(* Logix 5000 project; controller cal1632 1756-L62 rev 16.20; software revision 16.05; part 17 of 61 *)
(* tags used below, declared in another part *)
   FAULT : BOOL;
   p01_param_oven_timer_presets : DINT[32];
   p01_param_process_air_hl : REAL;
   p01_sys_enc : SYS_ENC;
   p01_sys_lc : Limit_Clamp;
   p01r09_pb_global_reset : BOOL;
   p02_real_from_hmi : hmi_real;
   p12_di_burner_auto : BOOL;
   p12_di_burner_safeties_ok : BOOL;
   p12_di_exh_flow_ok : BOOL;
   p12_di_flame_on : BOOL;
   p12_di_recirc_flow_ok : BOOL;
   p12_dint_to_hmi : DINT[16];
   p12_param_fast_to_soak : REAL;
   p12_param_lfl_hhl : REAL;
   p12_param_lfl_hl : REAL;
   p12_param_pid1_ff : REAL;
   p12_param_pid1_kd : REAL;
   p12_param_pid1_ki : REAL;
   p12_param_pid1_kp : REAL;
   p12_param_pid2_ff : REAL;
   p12_param_pid2_kd : REAL;
   p12_param_pid2_ki : REAL;
   p12_param_pid2_kp : REAL;
   p12_param_shutdown_temp : REAL;
   p12_param_soak_to_fast : REAL;
   p12_param_tc01_dev : REAL;
   p12_param_tc01_hl : REAL;
   p12_param_tc01z : REAL;
   p12_param_tc02z : REAL;
   p12_param_zone_pressure : REAL;
   p12r02 : routine;
   p12r02_shutdown_temp : BOOL;
   p12r02_timer_safe_temp : TIMER[2];
   p12r02_timer_warning : TIMER[4];
   p12r08 : routine;
   p12r08_timer_fault : TIMER[4];
   p12r08_timer_warning : TIMER[4];
   p12r09 : routine;
   p12r09_timer_fault : TIMER[4];
   p12r09_timer_warning : TIMER[8];
   p12r10 : routine;
   p12r10_timer_fault : TIMER[4];
   p12r10_timer_warning : TIMER[4];
   p12r20 : routine;
   p12r20_safeties_ok : BOOL;
   p12r20_state : DINT;
   p12r20_status : DINT;
   p12r20_timer_fault : TIMER[4];
   p12r20_timer_state_11 : TIMER;
   p12r20_timer_state_3 : TIMER;
   p12r20_timer_state_4 : TIMER;
   p12r20_timer_state_7 : TIMER;
   p12r20_timer_warning : TIMER[4];
   p12r30 : routine;
   p12r30_cv_man_sp : REAL;
   p12r30_request_heat : BOOL;
   p12r30_request_manual : BOOL;
   p12r30_request_soak_control : BOOL;
   p12r30_temp_deviation_setpoint : DINT;
   p12r30_timer_fault : TIMER[16];
   p12r30_timer_warning : TIMER[12];
   p12r31 : routine;
   p12r31_timer_fault : TIMER[5];
   p12r31_timer_warning : TIMER[5];
   p12r32 : routine;
   p12r32_timer_fault : TIMER[5];
   p12r32_timer_warning : TIMER[5];
(* P12_Zone_2, continued *)

ROUTINE R08_Warnings   (* ladder *)
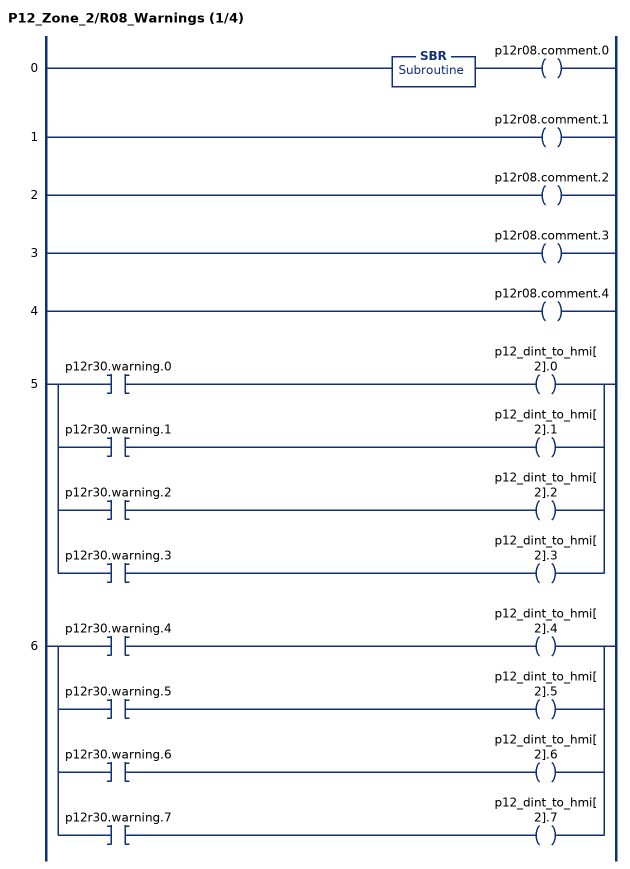
   0: SBR()OTE(p12r08.comment.0);
   1: OTE(p12r08.comment.1);
   2: OTE(p12r08.comment.2);
   3: OTE(p12r08.comment.3);
   4: OTE(p12r08.comment.4);
   5: [XIC(p12r30.warning.0) OTE(p12_dint_to_hmi[2].0) ,XIC(p12r30.warning.1) OTE(p12_dint_to_hmi[2].1) ,XIC(p12r30.warning.2) OTE(p12_dint_to_hmi[2].2) ,XIC(p12r30.warning.3) OTE(p12_dint_to_hmi[2].3) ];
   6: [XIC(p12r30.warning.4) OTE(p12_dint_to_hmi[2].4) ,XIC(p12r30.warning.5) OTE(p12_dint_to_hmi[2].5) ,XIC(p12r30.warning.6) OTE(p12_dint_to_hmi[2].6) ,XIC(p12r30.warning.7) OTE(p12_dint_to_hmi[2].7) ];
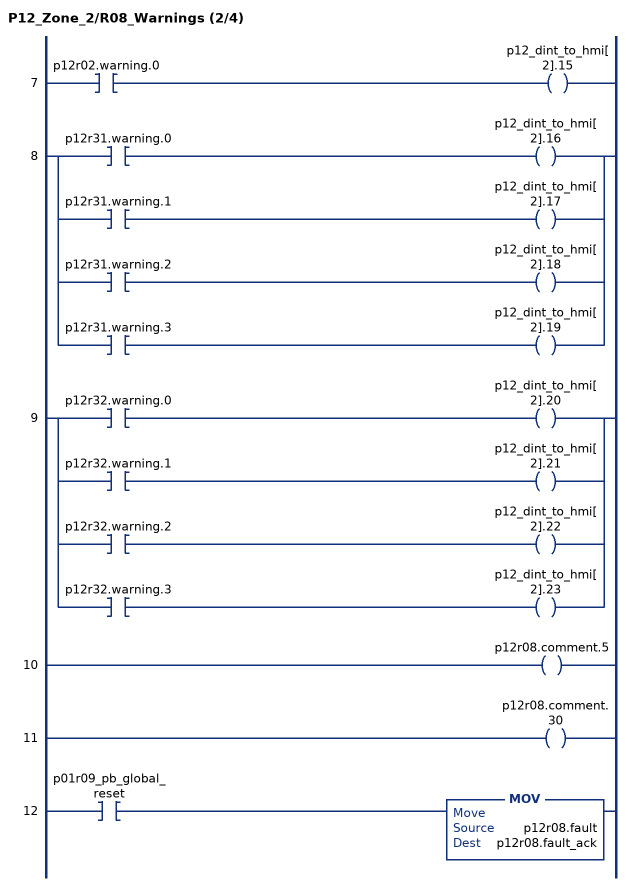
   7: XIC(p12r02.warning.0)OTE(p12_dint_to_hmi[2].15);
   8: [XIC(p12r31.warning.0) OTE(p12_dint_to_hmi[2].16) ,XIC(p12r31.warning.1) OTE(p12_dint_to_hmi[2].17) ,XIC(p12r31.warning.2) OTE(p12_dint_to_hmi[2].18) ,XIC(p12r31.warning.3) OTE(p12_dint_to_hmi[2].19) ];
   9: [XIC(p12r32.warning.0) OTE(p12_dint_to_hmi[2].20) ,XIC(p12r32.warning.1) OTE(p12_dint_to_hmi[2].21) ,XIC(p12r32.warning.2) OTE(p12_dint_to_hmi[2].22) ,XIC(p12r32.warning.3) OTE(p12_dint_to_hmi[2].23) ];
   10: OTE(p12r08.comment.5);
   11: OTE(p12r08.comment.30);
   12: XIC(p01r09_pb_global_reset)MOV(p12r08.fault,p12r08.fault_ack);
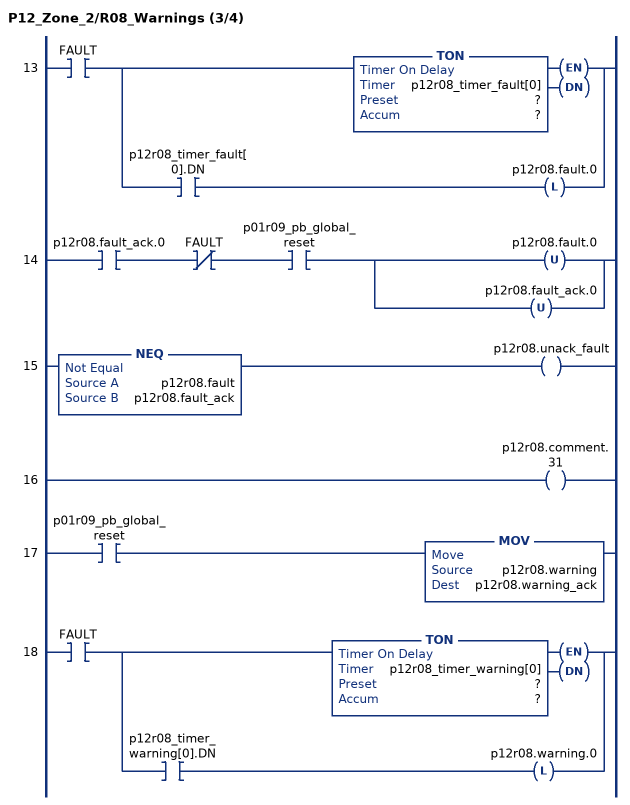
   13: XIC(FAULT)[TON(p12r08_timer_fault[0],?,?) ,XIC(p12r08_timer_fault[0].DN) OTL(p12r08.fault.0) ];
   14: XIC(p12r08.fault_ack.0)XIO(FAULT)XIC(p01r09_pb_global_reset)[OTU(p12r08.fault.0) ,OTU(p12r08.fault_ack.0) ];
   15: NEQ(p12r08.fault,p12r08.fault_ack)OTE(p12r08.unack_fault);
   16: OTE(p12r08.comment.31);
   17: XIC(p01r09_pb_global_reset)MOV(p12r08.warning,p12r08.warning_ack);
   18: XIC(FAULT)[TON(p12r08_timer_warning[0],?,?) ,XIC(p12r08_timer_warning[0].DN) OTL(p12r08.warning.0) ];
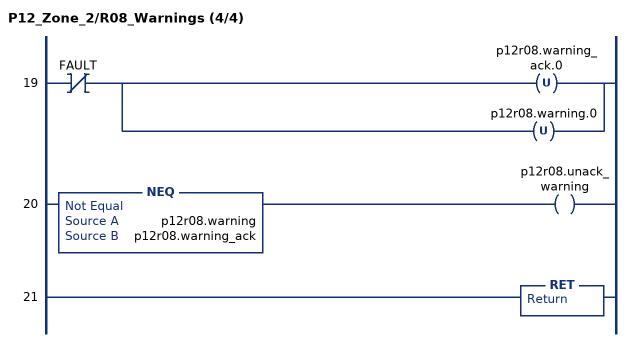
   19: XIO(FAULT)[OTU(p12r08.warning_ack.0) ,OTU(p12r08.warning.0) ];
   20: NEQ(p12r08.warning,p12r08.warning_ack)OTE(p12r08.unack_warning);
   21: RET();
END_ROUTINE

ROUTINE R09_Modes   (* ladder *)
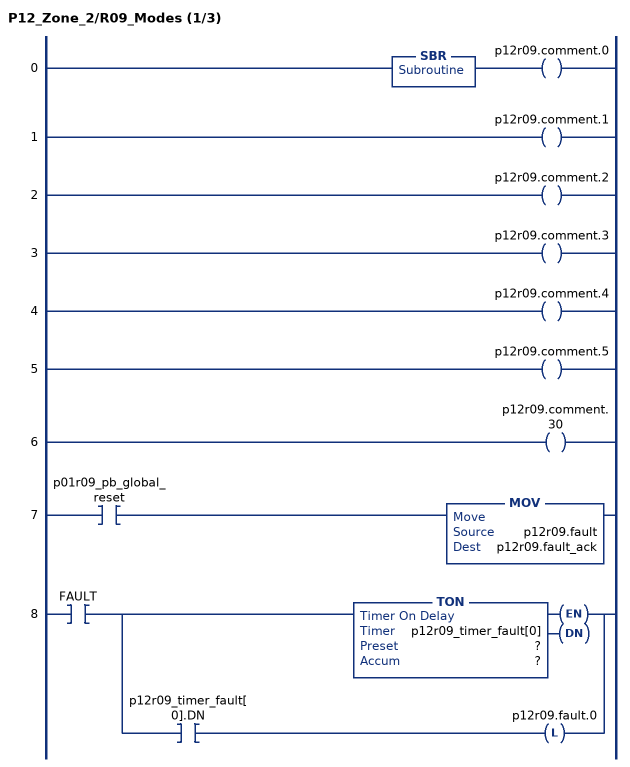
   0: SBR()OTE(p12r09.comment.0);
   1: OTE(p12r09.comment.1);
   2: OTE(p12r09.comment.2);
   3: OTE(p12r09.comment.3);
   4: OTE(p12r09.comment.4);
   5: OTE(p12r09.comment.5);
   6: OTE(p12r09.comment.30);
   7: XIC(p01r09_pb_global_reset)MOV(p12r09.fault,p12r09.fault_ack);
   8: XIC(FAULT)[TON(p12r09_timer_fault[0],?,?) ,XIC(p12r09_timer_fault[0].DN) OTL(p12r09.fault.0) ];
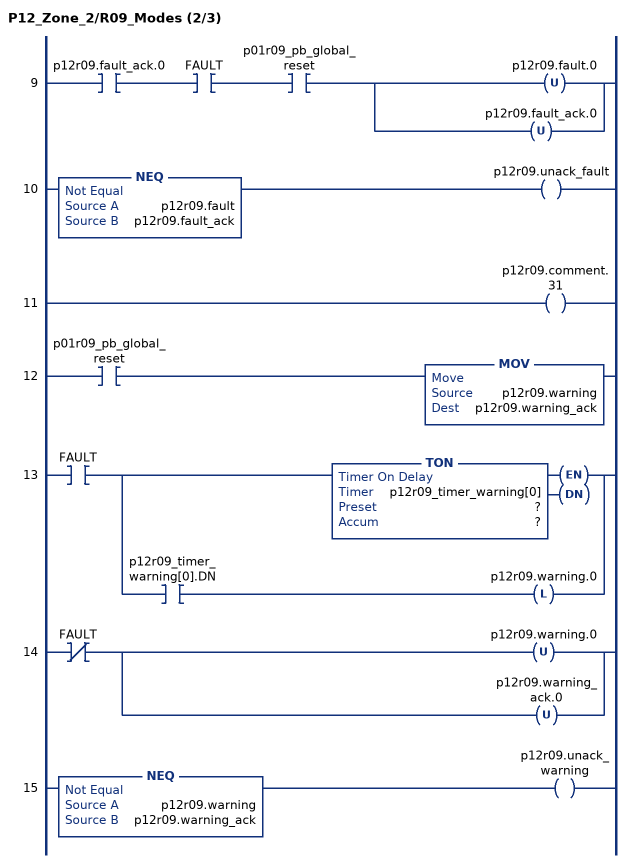
   9: XIC(p12r09.fault_ack.0)XIC(FAULT)XIC(p01r09_pb_global_reset)[OTU(p12r09.fault.0) ,OTU(p12r09.fault_ack.0) ];
   10: NEQ(p12r09.fault,p12r09.fault_ack)OTE(p12r09.unack_fault);
   11: OTE(p12r09.comment.31);
   12: XIC(p01r09_pb_global_reset)MOV(p12r09.warning,p12r09.warning_ack);
   13: XIC(FAULT)[TON(p12r09_timer_warning[0],?,?) ,XIC(p12r09_timer_warning[0].DN) OTL(p12r09.warning.0) ];
   14: XIO(FAULT)[OTU(p12r09.warning.0) ,OTU(p12r09.warning_ack.0) ];
   15: NEQ(p12r09.warning,p12r09.warning_ack)OTE(p12r09.unack_warning);
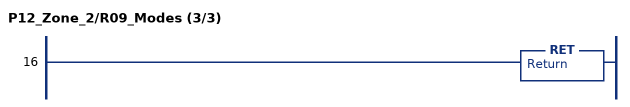
   16: RET();
END_ROUTINE

ROUTINE R10_Parameters   (* ladder *)
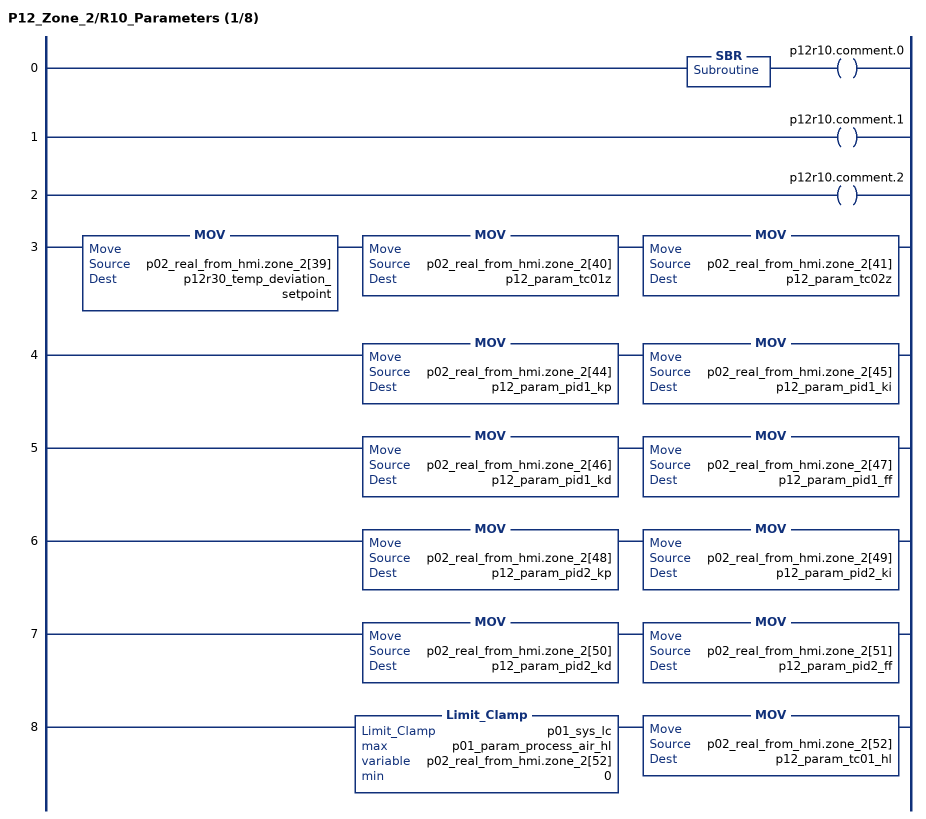
   0: SBR()OTE(p12r10.comment.0);
   1: OTE(p12r10.comment.1);
   2: OTE(p12r10.comment.2);
   3: MOV(p02_real_from_hmi.zone_2[39],p12r30_temp_deviation_setpoint)MOV(p02_real_from_hmi.zone_2[40],p12_param_tc01z)MOV(p02_real_from_hmi.zone_2[41],p12_param_tc02z);
   4: MOV(p02_real_from_hmi.zone_2[44],p12_param_pid1_kp)MOV(p02_real_from_hmi.zone_2[45],p12_param_pid1_ki);
   5: MOV(p02_real_from_hmi.zone_2[46],p12_param_pid1_kd)MOV(p02_real_from_hmi.zone_2[47],p12_param_pid1_ff);
   6: MOV(p02_real_from_hmi.zone_2[48],p12_param_pid2_kp)MOV(p02_real_from_hmi.zone_2[49],p12_param_pid2_ki);
   7: MOV(p02_real_from_hmi.zone_2[50],p12_param_pid2_kd)MOV(p02_real_from_hmi.zone_2[51],p12_param_pid2_ff);
   8: Limit_Clamp(p01_sys_lc,p01_param_process_air_hl,p02_real_from_hmi.zone_2[52],0)MOV(p02_real_from_hmi.zone_2[52],p12_param_tc01_hl);
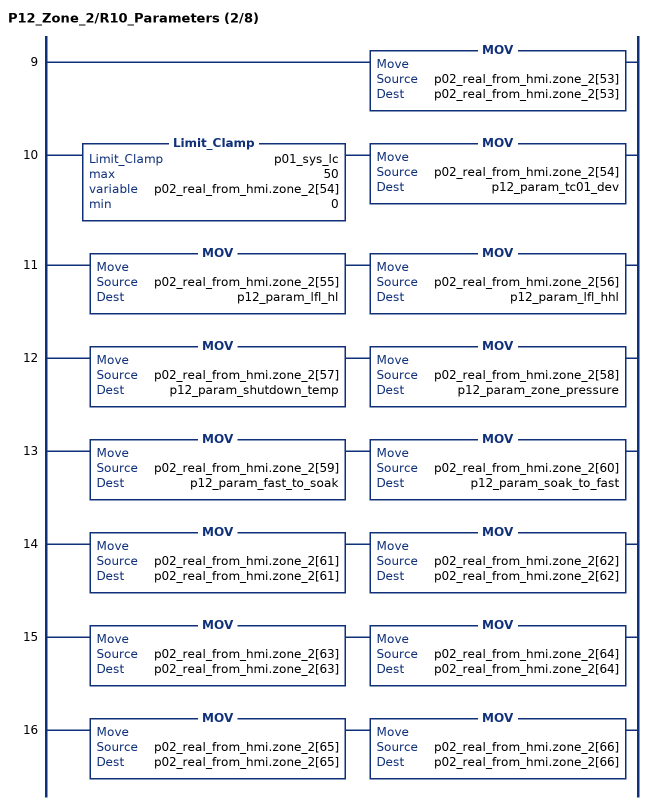
   9: MOV(p02_real_from_hmi.zone_2[53],p02_real_from_hmi.zone_2[53]);
   10: Limit_Clamp(p01_sys_lc,50,p02_real_from_hmi.zone_2[54],0)MOV(p02_real_from_hmi.zone_2[54],p12_param_tc01_dev);
   11: MOV(p02_real_from_hmi.zone_2[55],p12_param_lfl_hl)MOV(p02_real_from_hmi.zone_2[56],p12_param_lfl_hhl);
   12: MOV(p02_real_from_hmi.zone_2[57],p12_param_shutdown_temp)MOV(p02_real_from_hmi.zone_2[58],p12_param_zone_pressure);
   13: MOV(p02_real_from_hmi.zone_2[59],p12_param_fast_to_soak)MOV(p02_real_from_hmi.zone_2[60],p12_param_soak_to_fast);
   14: MOV(p02_real_from_hmi.zone_2[61],p02_real_from_hmi.zone_2[61])MOV(p02_real_from_hmi.zone_2[62],p02_real_from_hmi.zone_2[62]);
   15: MOV(p02_real_from_hmi.zone_2[63],p02_real_from_hmi.zone_2[63])MOV(p02_real_from_hmi.zone_2[64],p02_real_from_hmi.zone_2[64]);
   16: MOV(p02_real_from_hmi.zone_2[65],p02_real_from_hmi.zone_2[65])MOV(p02_real_from_hmi.zone_2[66],p02_real_from_hmi.zone_2[66]);
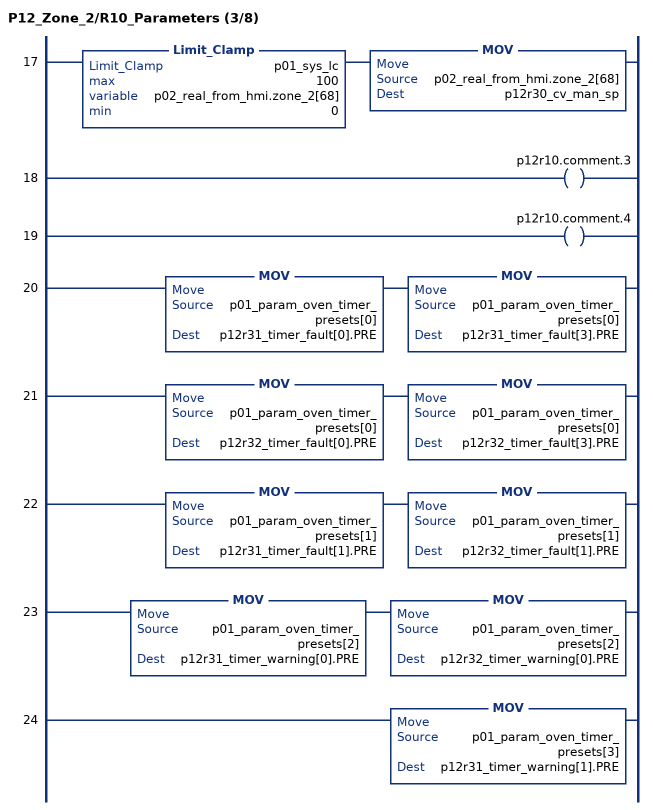
   17: Limit_Clamp(p01_sys_lc,100,p02_real_from_hmi.zone_2[68],0)MOV(p02_real_from_hmi.zone_2[68],p12r30_cv_man_sp);
   18: OTE(p12r10.comment.3);
   19: OTE(p12r10.comment.4);
   20: MOV(p01_param_oven_timer_presets[0],p12r31_timer_fault[0].PRE)MOV(p01_param_oven_timer_presets[0],p12r31_timer_fault[3].PRE);
   21: MOV(p01_param_oven_timer_presets[0],p12r32_timer_fault[0].PRE)MOV(p01_param_oven_timer_presets[0],p12r32_timer_fault[3].PRE);
   22: MOV(p01_param_oven_timer_presets[1],p12r31_timer_fault[1].PRE)MOV(p01_param_oven_timer_presets[1],p12r32_timer_fault[1].PRE);
   23: MOV(p01_param_oven_timer_presets[2],p12r31_timer_warning[0].PRE)MOV(p01_param_oven_timer_presets[2],p12r32_timer_warning[0].PRE);
   24: MOV(p01_param_oven_timer_presets[3],p12r31_timer_warning[1].PRE);
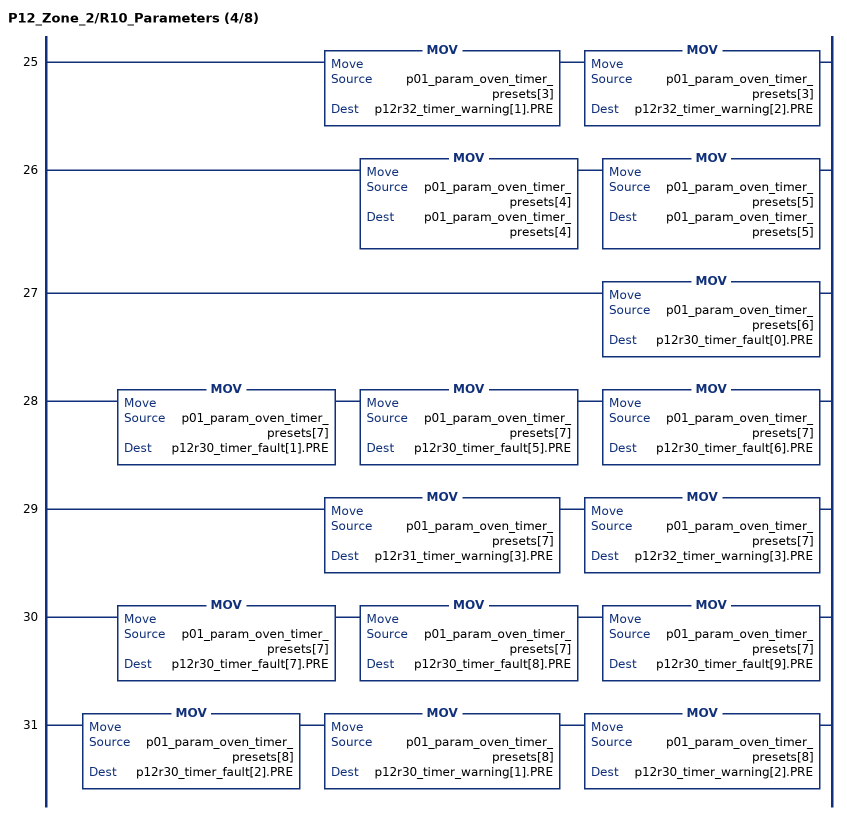
   25: MOV(p01_param_oven_timer_presets[3],p12r32_timer_warning[1].PRE)MOV(p01_param_oven_timer_presets[3],p12r32_timer_warning[2].PRE);
   26: MOV(p01_param_oven_timer_presets[4],p01_param_oven_timer_presets[4])MOV(p01_param_oven_timer_presets[5],p01_param_oven_timer_presets[5]);
   27: MOV(p01_param_oven_timer_presets[6],p12r30_timer_fault[0].PRE);
   28: MOV(p01_param_oven_timer_presets[7],p12r30_timer_fault[1].PRE)MOV(p01_param_oven_timer_presets[7],p12r30_timer_fault[5].PRE)MOV(p01_param_oven_timer_presets[7],p12r30_timer_fault[6].PRE);
   29: MOV(p01_param_oven_timer_presets[7],p12r31_timer_warning[3].PRE)MOV(p01_param_oven_timer_presets[7],p12r32_timer_warning[3].PRE);
   30: MOV(p01_param_oven_timer_presets[7],p12r30_timer_fault[7].PRE)MOV(p01_param_oven_timer_presets[7],p12r30_timer_fault[8].PRE)MOV(p01_param_oven_timer_presets[7],p12r30_timer_fault[9].PRE);
   31: MOV(p01_param_oven_timer_presets[8],p12r30_timer_fault[2].PRE)MOV(p01_param_oven_timer_presets[8],p12r30_timer_warning[1].PRE)MOV(p01_param_oven_timer_presets[8],p12r30_timer_warning[2].PRE);
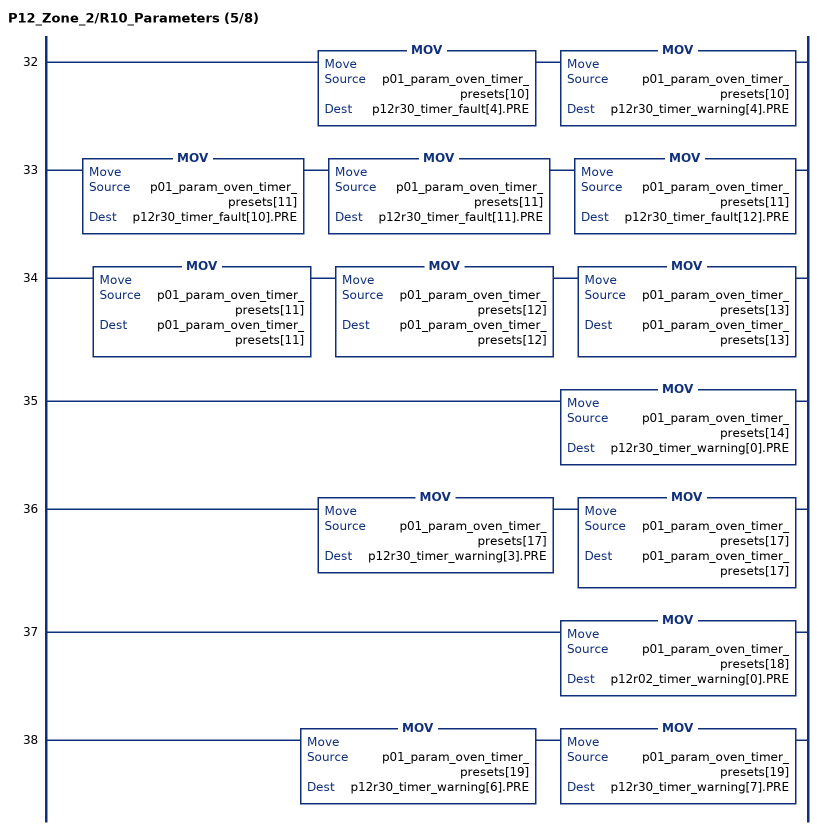
   32: MOV(p01_param_oven_timer_presets[10],p12r30_timer_fault[4].PRE)MOV(p01_param_oven_timer_presets[10],p12r30_timer_warning[4].PRE);
   33: MOV(p01_param_oven_timer_presets[11],p12r30_timer_fault[10].PRE)MOV(p01_param_oven_timer_presets[11],p12r30_timer_fault[11].PRE)MOV(p01_param_oven_timer_presets[11],p12r30_timer_fault[12].PRE);
   34: MOV(p01_param_oven_timer_presets[11],p01_param_oven_timer_presets[11])MOV(p01_param_oven_timer_presets[12],p01_param_oven_timer_presets[12])MOV(p01_param_oven_timer_presets[13],p01_param_oven_timer_presets[13]);
   35: MOV(p01_param_oven_timer_presets[14],p12r30_timer_warning[0].PRE);
   36: MOV(p01_param_oven_timer_presets[17],p12r30_timer_warning[3].PRE)MOV(p01_param_oven_timer_presets[17],p01_param_oven_timer_presets[17]);
   37: MOV(p01_param_oven_timer_presets[18],p12r02_timer_warning[0].PRE);
   38: MOV(p01_param_oven_timer_presets[19],p12r30_timer_warning[6].PRE)MOV(p01_param_oven_timer_presets[19],p12r30_timer_warning[7].PRE);
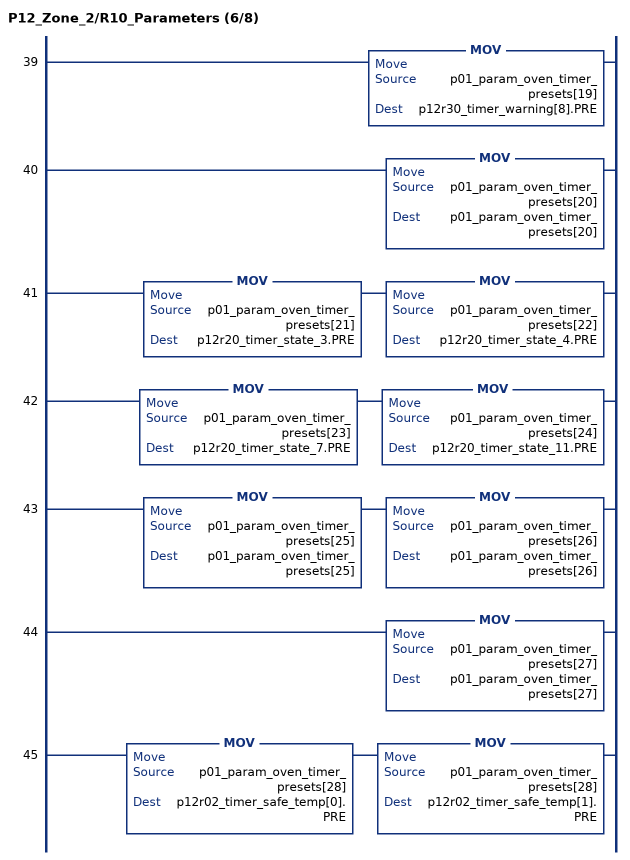
   39: MOV(p01_param_oven_timer_presets[19],p12r30_timer_warning[8].PRE);
   40: MOV(p01_param_oven_timer_presets[20],p01_param_oven_timer_presets[20]);
   41: MOV(p01_param_oven_timer_presets[21],p12r20_timer_state_3.PRE)MOV(p01_param_oven_timer_presets[22],p12r20_timer_state_4.PRE);
   42: MOV(p01_param_oven_timer_presets[23],p12r20_timer_state_7.PRE)MOV(p01_param_oven_timer_presets[24],p12r20_timer_state_11.PRE);
   43: MOV(p01_param_oven_timer_presets[25],p01_param_oven_timer_presets[25])MOV(p01_param_oven_timer_presets[26],p01_param_oven_timer_presets[26]);
   44: MOV(p01_param_oven_timer_presets[27],p01_param_oven_timer_presets[27]);
   45: MOV(p01_param_oven_timer_presets[28],p12r02_timer_safe_temp[0].PRE)MOV(p01_param_oven_timer_presets[28],p12r02_timer_safe_temp[1].PRE);
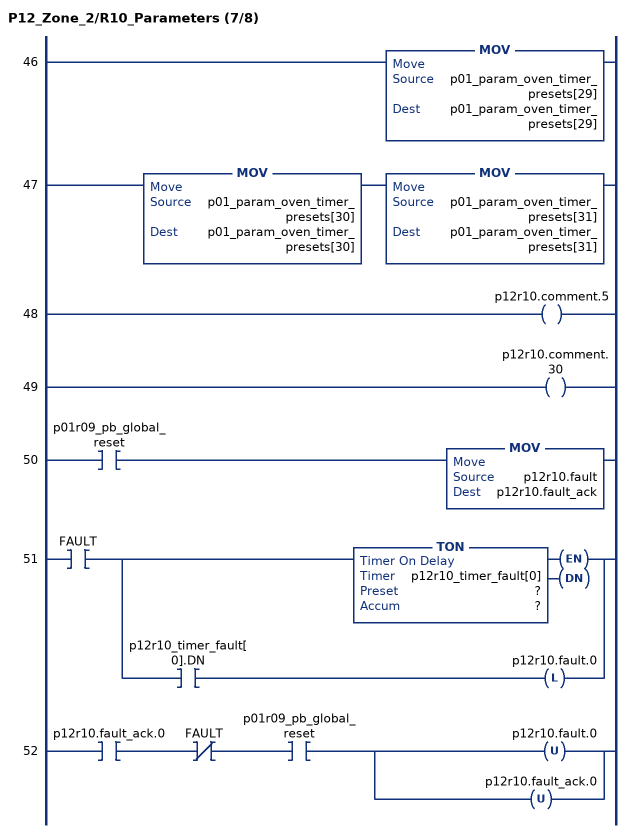
   46: MOV(p01_param_oven_timer_presets[29],p01_param_oven_timer_presets[29]);
   47: MOV(p01_param_oven_timer_presets[30],p01_param_oven_timer_presets[30])MOV(p01_param_oven_timer_presets[31],p01_param_oven_timer_presets[31]);
   48: OTE(p12r10.comment.5);
   49: OTE(p12r10.comment.30);
   50: XIC(p01r09_pb_global_reset)MOV(p12r10.fault,p12r10.fault_ack);
   51: XIC(FAULT)[TON(p12r10_timer_fault[0],?,?) ,XIC(p12r10_timer_fault[0].DN) OTL(p12r10.fault.0) ];
   52: XIC(p12r10.fault_ack.0)XIO(FAULT)XIC(p01r09_pb_global_reset)[OTU(p12r10.fault.0) ,OTU(p12r10.fault_ack.0) ];
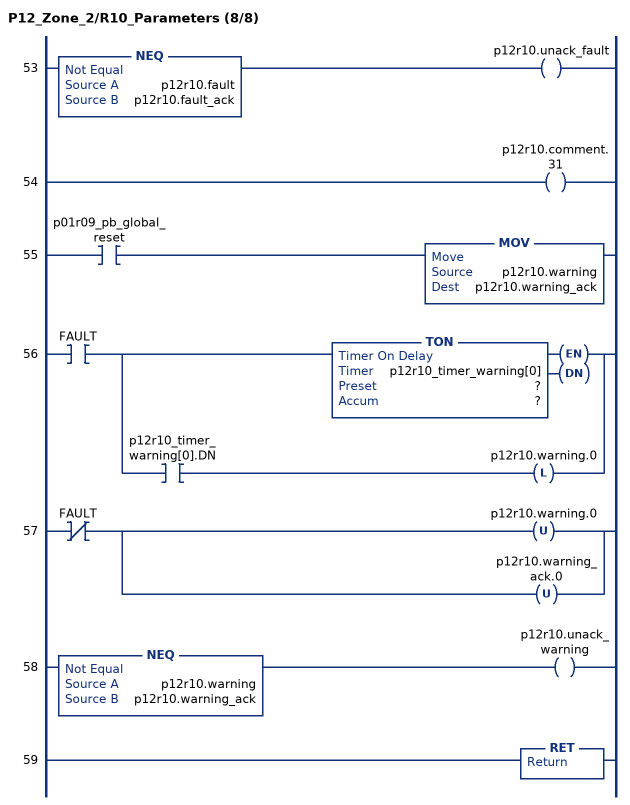
   53: NEQ(p12r10.fault,p12r10.fault_ack)OTE(p12r10.unack_fault);
   54: OTE(p12r10.comment.31);
   55: XIC(p01r09_pb_global_reset)MOV(p12r10.warning,p12r10.warning_ack);
   56: XIC(FAULT)[TON(p12r10_timer_warning[0],?,?) ,XIC(p12r10_timer_warning[0].DN) OTL(p12r10.warning.0) ];
   57: XIO(FAULT)[OTU(p12r10.warning.0) ,OTU(p12r10.warning_ack.0) ];
   58: NEQ(p12r10.warning,p12r10.warning_ack)OTE(p12r10.unack_warning);
   59: RET();
END_ROUTINE

ROUTINE R20_Temp_Sequence   (* ladder *)
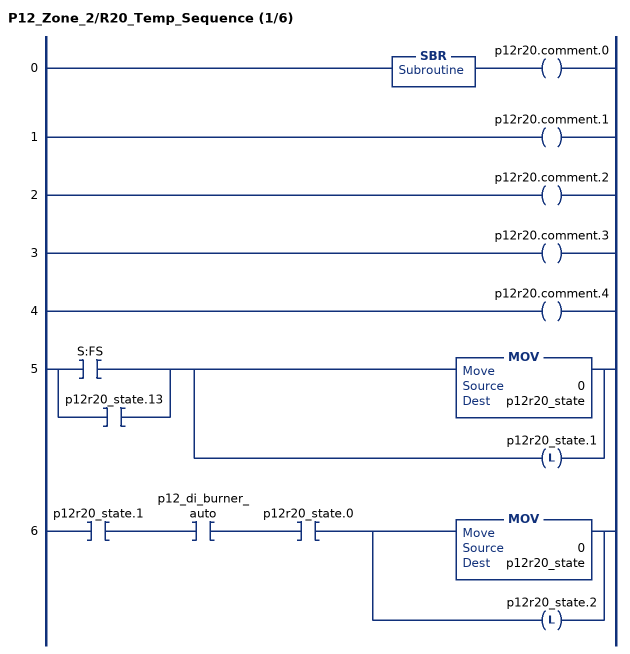
   0: SBR()OTE(p12r20.comment.0);
   1: OTE(p12r20.comment.1);
   2: OTE(p12r20.comment.2);
   3: OTE(p12r20.comment.3);
   4: OTE(p12r20.comment.4);
   5: [XIC(S:FS) ,XIC(p12r20_state.13) ][MOV(0,p12r20_state) ,OTL(p12r20_state.1) ];
   6: XIC(p12r20_state.1)XIC(p12_di_burner_auto)XIC(p12r20_state.0)[MOV(0,p12r20_state) ,OTL(p12r20_state.2) ];
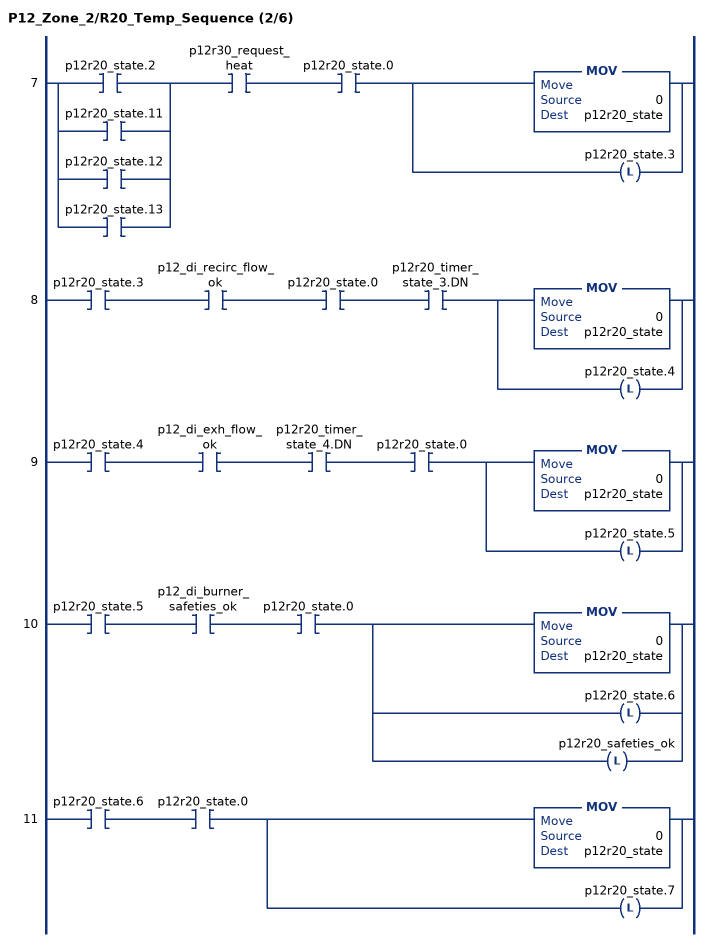
   7: [XIC(p12r20_state.2) ,XIC(p12r20_state.11) ,XIC(p12r20_state.12) ,XIC(p12r20_state.13) ]XIC(p12r30_request_heat)XIC(p12r20_state.0)[MOV(0,p12r20_state) ,OTL(p12r20_state.3) ];
   8: XIC(p12r20_state.3)XIC(p12_di_recirc_flow_ok)XIC(p12r20_state.0)XIC(p12r20_timer_state_3.DN)[MOV(0,p12r20_state) ,OTL(p12r20_state.4) ];
   9: XIC(p12r20_state.4)XIC(p12_di_exh_flow_ok)XIC(p12r20_timer_state_4.DN)XIC(p12r20_state.0)[MOV(0,p12r20_state) ,OTL(p12r20_state.5) ];
   10: XIC(p12r20_state.5)XIC(p12_di_burner_safeties_ok)XIC(p12r20_state.0)[MOV(0,p12r20_state) ,OTL(p12r20_state.6) ,OTL(p12r20_safeties_ok) ];
   11: XIC(p12r20_state.6)XIC(p12r20_state.0)[MOV(0,p12r20_state) ,OTL(p12r20_state.7) ];
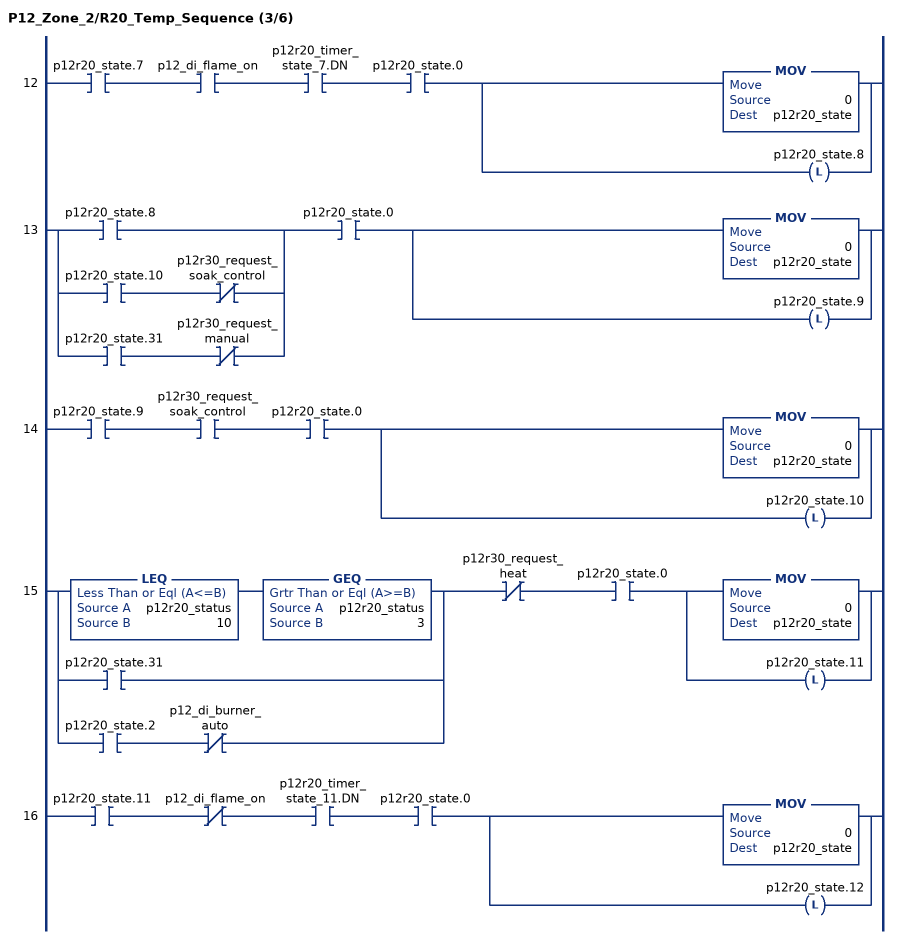
   12: XIC(p12r20_state.7)XIC(p12_di_flame_on)XIC(p12r20_timer_state_7.DN)XIC(p12r20_state.0)[MOV(0,p12r20_state) ,OTL(p12r20_state.8) ];
   13: [XIC(p12r20_state.8) ,XIC(p12r20_state.10) XIO(p12r30_request_soak_control) ,XIC(p12r20_state.31) XIO(p12r30_request_manual) ]XIC(p12r20_state.0)[MOV(0,p12r20_state) ,OTL(p12r20_state.9) ];
   14: XIC(p12r20_state.9)XIC(p12r30_request_soak_control)XIC(p12r20_state.0)[MOV(0,p12r20_state) ,OTL(p12r20_state.10) ];
   15: [[LEQ(p12r20_status,10) GEQ(p12r20_status,3) ,XIC(p12r20_state.31) ] ,XIC(p12r20_state.2) XIO(p12_di_burner_auto) ]XIO(p12r30_request_heat)XIC(p12r20_state.0)[MOV(0,p12r20_state) ,OTL(p12r20_state.11) ];
   16: XIC(p12r20_state.11)XIO(p12_di_flame_on)XIC(p12r20_timer_state_11.DN)XIC(p12r20_state.0)[MOV(0,p12r20_state) ,OTL(p12r20_state.12) ];
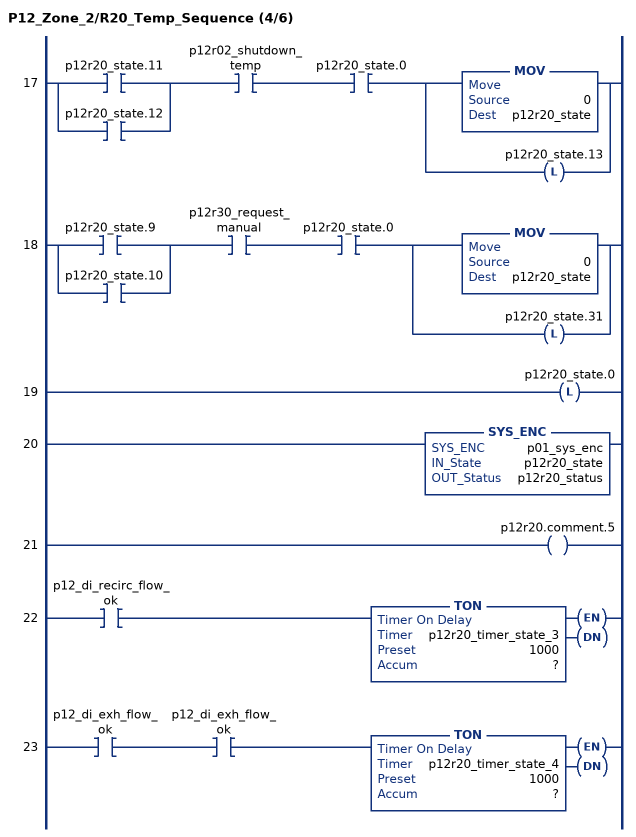
   17: [XIC(p12r20_state.11) ,XIC(p12r20_state.12) ]XIC(p12r02_shutdown_temp)XIC(p12r20_state.0)[MOV(0,p12r20_state) ,OTL(p12r20_state.13) ];
   18: [XIC(p12r20_state.9) ,XIC(p12r20_state.10) ]XIC(p12r30_request_manual)XIC(p12r20_state.0)[MOV(0,p12r20_state) ,OTL(p12r20_state.31) ];
   19: OTL(p12r20_state.0);
   20: SYS_ENC(p01_sys_enc,p12r20_state,p12r20_status);
   21: OTE(p12r20.comment.5);
   22: XIC(p12_di_recirc_flow_ok)TON(p12r20_timer_state_3,?,?);
   23: XIC(p12_di_exh_flow_ok)XIC(p12_di_exh_flow_ok)TON(p12r20_timer_state_4,?,?);
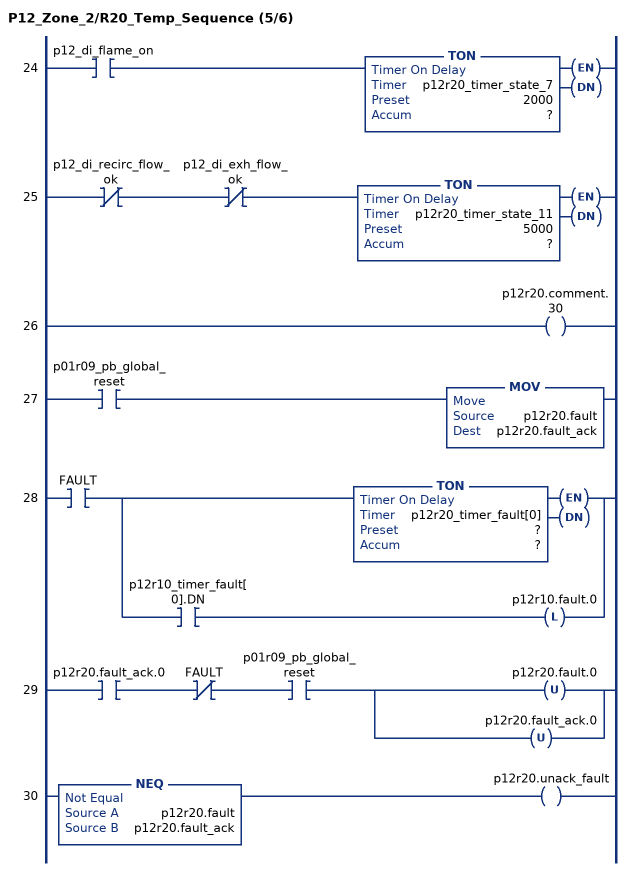
   24: XIC(p12_di_flame_on)TON(p12r20_timer_state_7,?,?);
   25: XIO(p12_di_recirc_flow_ok)XIO(p12_di_exh_flow_ok)TON(p12r20_timer_state_11,?,?);
   26: OTE(p12r20.comment.30);
   27: XIC(p01r09_pb_global_reset)MOV(p12r20.fault,p12r20.fault_ack);
   28: XIC(FAULT)[TON(p12r20_timer_fault[0],?,?) ,XIC(p12r10_timer_fault[0].DN) OTL(p12r10.fault.0) ];
   29: XIC(p12r20.fault_ack.0)XIO(FAULT)XIC(p01r09_pb_global_reset)[OTU(p12r20.fault.0) ,OTU(p12r20.fault_ack.0) ];
   30: NEQ(p12r20.fault,p12r20.fault_ack)OTE(p12r20.unack_fault);
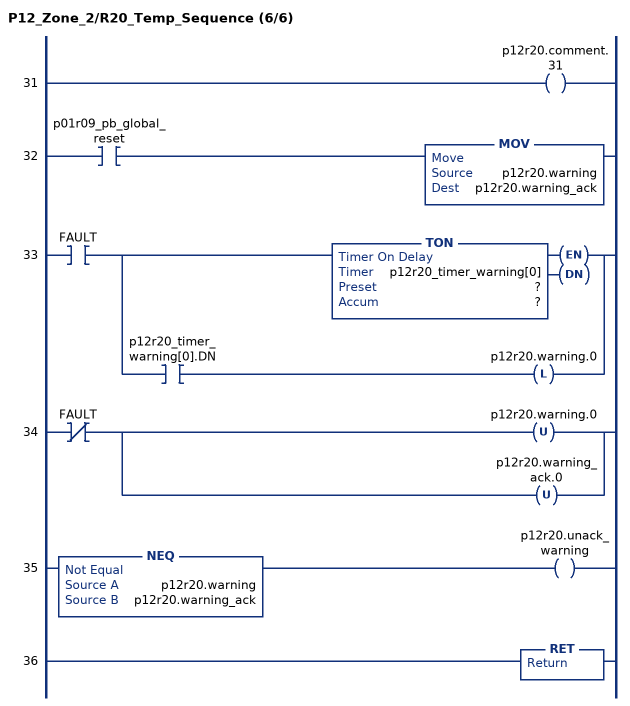
   31: OTE(p12r20.comment.31);
   32: XIC(p01r09_pb_global_reset)MOV(p12r20.warning,p12r20.warning_ack);
   33: XIC(FAULT)[TON(p12r20_timer_warning[0],?,?) ,XIC(p12r20_timer_warning[0].DN) OTL(p12r20.warning.0) ];
   34: XIO(FAULT)[OTU(p12r20.warning.0) ,OTU(p12r20.warning_ack.0) ];
   35: NEQ(p12r20.warning,p12r20.warning_ack)OTE(p12r20.unack_warning);
   36: RET();
END_ROUTINE
